Fanuc KAREL source: V_RUN_FIND.kl

PROGRAM T
%NOLOCKGROUP
VAR
 v0 : STRING[40]
 v1 : INTEGER
 v2 : INTEGER
BEGIN
 V_RUN_FIND(v0, v1, v2)
END T
